# EPICS substitutions: pimegaApp/Db/pimega540d.substitutions
file "pimega.template" {
  {}
}

file "module.template" {
   pattern { MODULE, ADDR }
           { M1:,    0    }
           { M2:,    1    }
           { M3:,    2    }
           { M4:,    3    }
}
